(* IEC 61131-3 sources: Industry-PLC-LLM/data/PLCBEAD_repo/PLCBEAD_PLCEmbed-main/PLC-BEAD/Source/GEB/DAY_OF_DATE, 1 file *)

(* ---- DAY_OF_DATE.ST ---- *)
FUNCTION DAY_OF_DATE:DINT
	VAR_INPUT
		IDATE :	UDINT;
	END_VAR

	DAY_OF_DATE := UDINT_TO_DINT(IDATE / UDINT#86400);
END_FUNCTION

PROGRAM program0
  VAR
    LocalVar0 : UDINT;
	LocalOUT  : DINT;
  END_VAR
  	LocalOUT := DAY_OF_DATE(LocalVar0);
END_PROGRAM
